(* PLC project Sin nombre, Desconocido Sin nombre 1 *)
(* stored: creationDateTime 2025-10-24T04:06:02, modificationDateTime 2025-10-26T05:05:52 *)

PROGRAM ciclo_principal
  VAR
    inclinado AT %IX0.0 : BOOL;
  END_VAR
  VAR
    ultimo_tilt : BOOL;
    conteo_tilt : INT;
    CTU1 : CTU;
    estado1 : BOOL;
    TON0 : TON;
    TON1 : TON;
    segmento_a : BOOL;
    segmento_b : BOOL;
    segmento_c : BOOL;
    segmento_d : BOOL;
    segmento_e : BOOL;
    segmento_f : BOOL;
    segmento_g : BOOL;
    parpadear_led : BOOL;
    TON2 : TON;
    TOF0 : TOF;
    CTU0 : CTU;
  END_VAR
  VAR  (* added by the conversion: wires and edge detectors of the diagram *)
    R_TRIG1 : R_TRIG;
    R_TRIG2 : R_TRIG;
  END_VAR

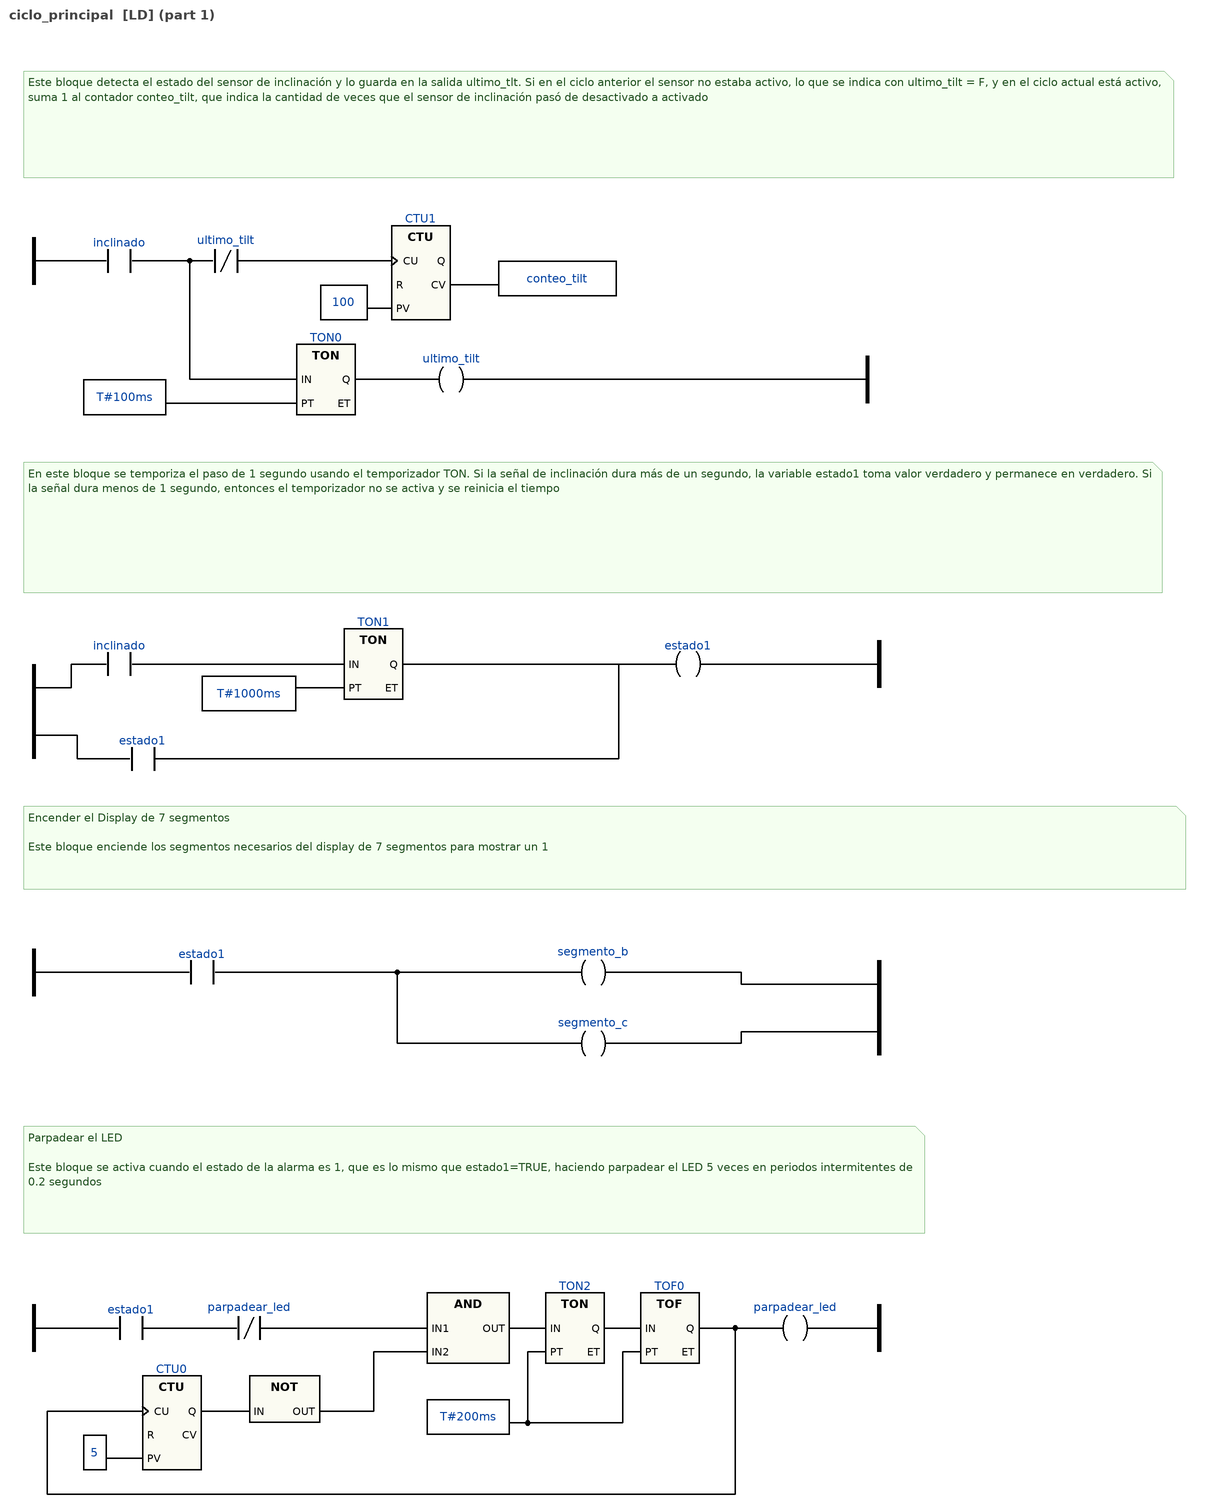
(* LD diagram, written out as Structured Text *)
(* Este bloque detecta el estado del sensor de inclinación y lo guarda en la salida ultimo_tlt. Si en el ciclo anterior el sensor no estaba activo, lo que se indica con ultimo_tilt = F, y en el ciclo actual está activo, suma 1 al contador conteo_tilt, que indica la cantidad de veces que el sensor de inclinación pasó de desactivado a activado *)
(* En este bloque se temporiza el paso de 1 segundo usando el temporizador TON. Si la señal de inclinación dura más de un segundo, la variable estado1 toma valor verdadero y permanece en verdadero. Si la señal dura menos de 1 segundo, entonces el temporizador no se activa y se reinicia el tiempo *)
TON1(IN := inclinado, PT := T#1000ms);
estado1 := estado1 OR TON1.Q;
TON0(IN := inclinado, PT := T#100ms);
ultimo_tilt := TON0.Q;
R_TRIG1(CLK := inclinado AND NOT ultimo_tilt);
CTU1(CU := R_TRIG1.Q, PV := 100);
conteo_tilt := CTU1.CV;
(* Encender el Display de 7 segmentos

Este bloque enciende los segmentos necesarios del display de 7 segmentos para mostrar un 1 *)
segmento_b := estado1;
segmento_c := estado1;
(* Parpadear el LED

Este bloque se activa cuando el estado de la alarma es 1, que es lo mismo que estado1=TRUE, haciendo parpadear el LED 5 veces en periodos intermitentes de 0.2 segundos *)
R_TRIG2(CLK := TOF0.Q);
CTU0(CU := R_TRIG2.Q, PV := 5);
TON2(IN := estado1 AND NOT parpadear_led AND NOT CTU0.Q, PT := T#200ms);
TOF0(IN := TON2.Q, PT := T#200ms);
parpadear_led := TOF0.Q;
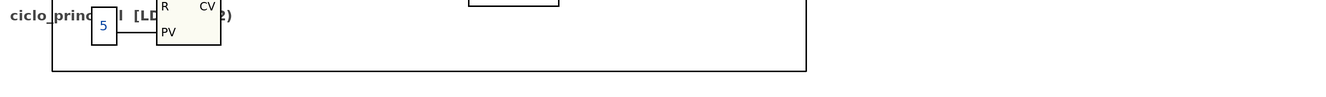
END_PROGRAM

CONFIGURATION Config0
  RESOURCE Res0 ON PLC
    TASK Principal(INTERVAL := T#200ms, PRIORITY := 0);
    PROGRAM registro_entradas WITH Principal : ciclo_principal;
  END_RESOURCE
END_CONFIGURATION
